(* Logix 5000 project; controller ListBoxToStringArray vendor 1 type 14 code 164 rev 38.11; software revision 38.01 *)

TASK MainTask (continuous, watchdog 500 ms) : MainProgram

MODULES
   Local : vendor 1 type 14 code 164 (ICP 4, rev 38.11)
END_MODULES

VAR_GLOBAL   (* controller tags *)
   SelectedString : STRING := 'E';
   StringsForListBox : STRING[10] := ([0] := 'A', [1] := 'B', [2] := 'C', [3] := 'D', [4] := 'E', [5] := 'F', [6] := 'G', [7] := 'H', [8] := 'I', [9] := 'J');
END_VAR

PROGRAM MainProgram   (* main routine MainRoutine *)

ROUTINE MainRoutine   (* ladder *)
END_ROUTINE
END_PROGRAM
